TYPE ST_NeedleChangeAllocateInfo :
STRUCT
	//確認是否要換
	CheckedChangeAllocate	:  BOOL;
	ChangeAllocate 			:  ARRAY[0..40] OF st_AllocationData;
END_STRUCT
END_TYPE

(* stored: Version 1.1.0.1, ProductVersion 3.1.4024.13
   DUT ST_NeedleChangeAllocateInfo: Id {299ea9cd-d7b9-4b43-aa7a-6d7dcac32f4b} *)
